{attribute 'linkalways'} 
{attribute 'no_explicit_call' := 'This FB is a CLASS and must be accessed using methods or properties'}
{attribute 'enable_dynamic_creation'}
FUNCTION_BLOCK FINAL OR_USINT EXTENDS Node
VAR
	in1 : _USINT(0);
	in2 : _USINT(0);
	out : _USINT(0);
END_VAR

METHOD PUBLIC Clone : I_Node
VAR
	pNode : POINTER TO OR_USINT;
END_VAR
pNode := __NEW(OR_USINT);
Clone := pNode^;
END_METHOD

METHOD FB_init : BOOL
VAR_INPUT
	bInitRetains : BOOL; // if TRUE, the retain variables are initialized (warm start / cold start)
	bInCopyCode : BOOL;  // if TRUE, the instance afterwards gets moved into the copy code (online change)
END_VAR
AddInput('in1',THIS^.in1);
AddInput('in2',THIS^.in2);
AddOutput('out', THIS^.out);
END_METHOD

METHOD PROTECTED OnExecute
VAR
END_VAR
out.Value := in1.Value OR in2.Value;
END_METHOD

END_FUNCTION_BLOCK

(* stored: Version 1.1.0.1, ProductVersion 3.1.4024.15
   POU OR_USINT: Id {93347483-f83e-4775-a18f-d465accc24da}, SpecialFunc None
   Folder Constructor: Id {d590a9bb-6bcc-40d2-b289-f3eeebe627f4}
   Method Clone: Id {a814ad18-cb48-4a50-86e5-203f4614783b}
   Method FB_init: Id {1e477580-1eb2-4890-a4f7-a569d94c8e6f}
   Method OnExecute: Id {925a8798-bac4-4d27-87ac-8b46ad1f67d3} *)
